Staubli VAL3: resumeProduct.pgx

program resumeProduct()
begin
  //暂停恢复
  if bPause
    bPause=false
    dioSet(io:doB_7_toolOn,1)
    if date:bWorTbMoving
      if dioGet(io:doB_9_tableOn)==0
        dioSet(io:doB_9_tableOn,1)
      endIf
    endIf
    restartMove()
  endIf
  //报警后处理
  if bSuspend==true
    bSuspend=false
    enablePower()
    read:bResumeCycle=true
    call production()
  endIf
end
